TYPE ST_MotionlinxAI_Controller_HMI :
	STRUCT
		Config	: ST_MotionlinxAI_Controller_Config;
		Command : ST_MotionlinxAI_Controller_Command;
		Status	: ST_MotionlinxAI_Controller_Status;
	END_STRUCT
END_TYPE

(* stored: Version 1.1.0.1, ProductVersion 3.1.4024.16
   DUT ST_MotionlinxAI_Controller_HMI: Id {0ddee52d-fdfc-4376-af9e-fc8cf071426b} *)
